RoboDK station: ME5286_Lab4_Serdoncillo_JustineJohnv1.rdk

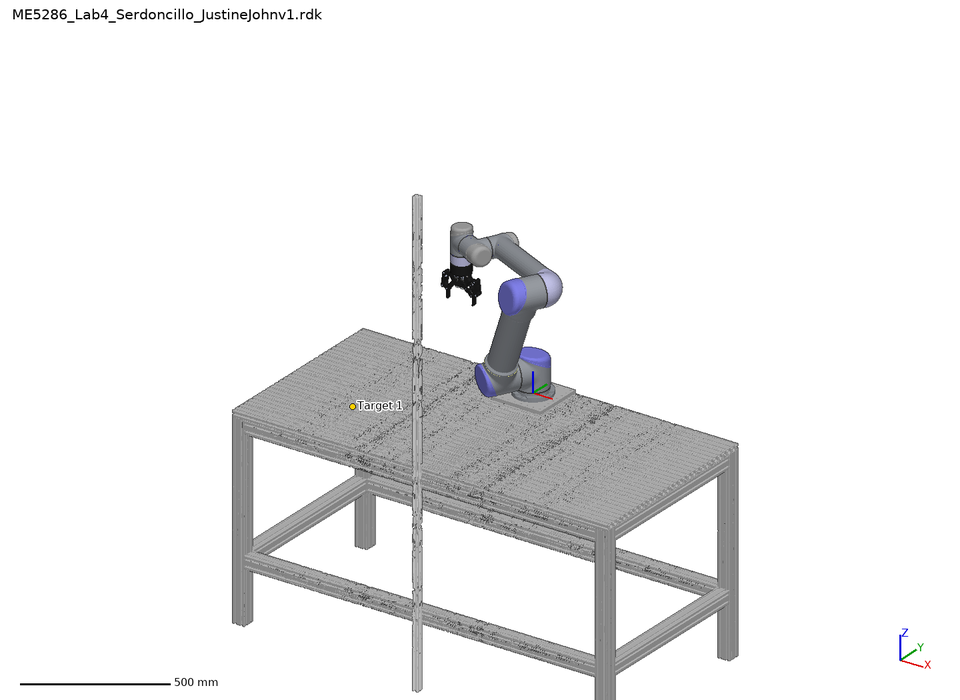
[picture v0: the station drawn from its stored meshes, robots at their saved joint values, targets as dots, program paths as lines]
Station ME5286_Lab4_Serdoncillo_JustineJohnv1 (saved by RoboDK 5.5.3). Poses are relative to the parent item; angles as X-Y-Z fixed-axis rotations.
  - frame UR5 Base at (0, 0, 0) mm
    - robot UR5: 6 axes, payload 5 kg, reach 850 mm, repeatability 0.1 mm, weight 18.4 kg
        modified DH rows (alpha deg, a mm, theta deg, d mm): 0, 0, 0, 89.2; 90, 0, 180, 0; 0, 425, 0, 0; 0, 392.43, 0, 109; -90, 0, 0, 93.65; 90, 0, 180, 82
        joint limits [-360, -360, -360, -360, -360, -360] to [360, 360, 360, 360, 360, 360]; home [0, -90, 90, 0, 90, 0]; saved at [-27.14, -115.32, 117.34, -92.04, -89.49, -26.91]
      - tool Gripper RobotiQ 85 Opened, TCP at (0, 0, 149.6) mm, size 147.4 x 146.8 x 75 mm
    - target Target 1 (Cartesian target) at (-388.22, -492.26, 39) mm, rotated rx 177.02 ry -0.73 rz 86.38 deg; joints [41.133, -63.138, 92.728, -116.961, -88.419, 44.733] of UR5
    - target Target 2 (Cartesian target) at (-388.22, -492.26, 39) mm, rotated rx -50 ry 58 rz -176 deg; joints [-116.508, -127.571, 233.195, -85.641, -85.367, -117.262] of UR5
  - object table_base_setup at (0, 0, 0) mm, rotated rx 0 ry 0 rz -90 deg, size 1524 x 762 x 800.1 mm, geometry from table_base_setup.STEP
  - object 6ft_beam_table at (0, -675, 1000) mm, size 25.4 x 25.4 x 1828.8 mm, geometry from 6ft_beam_table.IGS
  - Python program ME5286_Lab4_Task_Serdoncillo_JustineJohnv3 (listed below)

--- Python program ME5286_Lab4_Task_Serdoncillo_JustineJohnv3 ---
# This macro shows an example of running a program on the robot using the Python API (online programming)
# More information about the RoboDK API appears here:
# https://robodk.com/doc/en/RoboDK-API.html
import sys
sys.path.append("C:\RoboDK\Python")
#############################################################
from robolink import *    # API to communicate with RoboDK
from robodk import *      # robodk robotics toolbox
RDK = Robolink()
robot = RDK.ItemUserPick('Select a robot', ITEM_TYPE_ROBOT)
if not robot.Valid():
    raise Exception('No robot selected or available')
RUN_ON_ROBOT = False
if RDK.RunMode() != RUNMODE_SIMULATE:
    RUN_ON_ROBOT = False
if RUN_ON_ROBOT:
    # Connect to the robot using default IP
    success = robot.Connect() # Try to connect once
    status, status_msg = robot.ConnectedState()
    if status != ROBOTCOM_READY:
        # Stop if the connection did not succeed
        print(status_msg)
        raise Exception("Failed to connect: " + status_msg)
    # This will set to run the API programs on the robot and the simulator (online programming)
    RDK.setRunMode(RUNMODE_RUN_ROBOT)
joints_ref = robot.Joints()
target_ref = robot.Pose()
pos_ref = target_ref.Pos()
robot.setPoseFrame(robot.PoseFrame())
robot.setPoseTool(robot.PoseTool())
###################################################################
## JJ Code down below
import numpy as np
###################################################################
linspeed = [250]
linaccel = [200]
joispeed = [15]
joiaccel = [60]
robot.setSpeed(50) # Set linear speed in mm/s
robot.setAcceleration(100) # Set acceleration in mm/s
robot.setSpeedJoints(15) # Set joint speed in deg/s
robot.setAccelerationJoints(60) # Set joint accel in deg/s^2
robot.setZoneData(2) # Set blending radius in mm
##################################################################
gripper_force = [127,127,127,127]
gripper_speed = [ 50, 50, 50, 50]
pos = np.array([ [0, 0, 0, 0] , [0, 9, 6, 3] ]) * 25.4
##################################################################
# input values here
tray_og =  [-389.00 ,-494.00] # origin of the tray in x,y,z
chuck_og = [-322.00 ,  40.00] # origin of the chuck in x,y,z
#-388.22 ,-492.26
#-322.39 ,  39.89: old chuck_og and not centered
#-320.37 ,  39.9
#deg = [130,122,4] # ideal orientation
#deg = [-180,0,4] # from Lab 3 but hitting other components
#deg = [-176.79,-1.10,-89.55]
deg = [-180,0,-90]
tray_z  = np.array([39,50,43,38]) + 33 # Lab 3 has z=70 but these measurements s
chuck_z = np.array([140,185,225,227]) + 40 # 2 and 3 not sure

twist = [False,True,False,True]
#twist = [False, False, False, False]
#twist_num = [10,7]
twist_num = [6,3]
twist_torque = [3,2]
#############################################
theta_1 = 0
theta_2 = np.pi
cB = np.cos(theta_1)
sB = np.sin(theta_1)
cC = np.cos(theta_2)
sC = np.sin(theta_2)
TB = tray_og.copy()
TC = chuck_og.copy()
RTAB = np.array([[cB,-sB,TB[0]],[sB,cB,TB[1]],[0,0,1]])
RTAC = np.array([[cC,-sC,TC[0]],[sC,cC,TC[1]],[0,0,1]])

tray   = np.zeros((4,6))
chuck  = np.zeros((4,6))
tray[:,3] = deg[0]
tray[:,4] = deg[1]
tray[:,5] = deg[2]
chuck[:,0] = TC[0]
chuck[:,1] = TC[1]
chuck[:,3] = deg[0]
chuck[:,4] = deg[1]
chuck[:,5] = deg[2]
for j in range(4):
  P1B = np.array([[pos[0,j]],[pos[1,j]],[1]])
  P1A = RTAB @ P1B
  tray[j,0] = P1A[0]
  tray[j,1] = P1A[1]
  tray[j,2] = tray_z[j]
  chuck[j,2] = chuck_z[j]
tray_up = tray.copy()
tray_up[:,2] += 30
chuck_up = chuck.copy()
chuck_up[:,2] += 110

#twist_before = np.zeros((2,6))
'''
twist_before[0] = chuck[1]
twist_before[1] = chuck[3]
twist_after = twist_before.copy()
twist_after[:,5] = 90
'''
twist_before = [-27.14,-115.32,117.34,-92.04,-89.49,-206.91]
#twist_before[0] = [-27.14,-115.32,117.34,-92.04,-89.49,-206.91]
twist_after = twist_before.copy()
twist_after[5] += 180

twist_count = 0

###################################################################
''' Do manual stuff rn '''
home = [0, -90, 0, -90, 0, 0]
robot.MoveJ(home)
safe = [35.30,-90.35,87.92,-90.26,-90.32,-43.42]
robot.MoveJ(safe)

robot.RunCodeCustom('unclamp()',INSTRUCTION_INSERT_CODE)
#robot.RunCodeCustom('clamp()',INSTRUCTION_INSERT_CODE)
#range(4)

for i in np.arange(0,2):
    robot.RunCodeCustom('rq_set_force(%i)' %gripper_force[i], INSTRUCTION_CALL_PROGRAM)
    robot.RunCodeCustom('rq_set_speed(%i)' %gripper_speed[i], INSTRUCTION_CALL_PROGRAM)
    robot.MoveL(xyzrpw_2_pose(tray[i]))
    robot.RunCodeCustom('rq_close_and_wait()',INSTRUCTION_CALL_PROGRAM)
    robot.MoveL(xyzrpw_2_pose(tray_up[i]))
    robot.MoveL(xyzrpw_2_pose(chuck_up[i]))
    robot.MoveL(xyzrpw_2_pose(chuck[i]))
    #robot.RunCodeCustom('sleep(10)',INSTRUCTION_CALL_PROGRAM)
    if i != 3:
        robot.RunCodeCustom('rq_open_and_wait()',INSTRUCTION_CALL_PROGRAM)
    if twist[i] == True:
        for tnum in range(twist_num[twist_count]):
            robot.MoveJ(twist_before)
            #robot.MoveJ(xyzrpw_2_pose(twist_before[twist_count]))
            robot.RunCodeCustom('rq_close_and_wait()',INSTRUCTION_CALL_PROGRAM)
            robot.MoveJ(twist_after)
            #robot.MoveJ(xyzrpw_2_pose(twist_after[twist_count]))
            robot.RunCodeCustom('rq_open_and_wait()',INSTRUCTION_CALL_PROGRAM)
        robot.RunCodeCustom('tighten_torque(%i,0,1.57,2,2,1,100,100,50)' %twist_torque[twist_count],INSTRUCTION_INSERT_CODE)
        twist_count += 1
    if i == 0:
        robot.RunCodeCustom('clamp()',INSTRUCTION_INSERT_CODE)
    elif i == 3:
        robot.RunCodeCustom('unclamp()',INSTRUCTION_INSERT_CODE)
    robot.MoveL(xyzrpw_2_pose(chuck[i]))
    robot.MoveL(xyzrpw_2_pose(chuck_up[i]))
    #robot.RunCodeCustom('sleep(10)',INSTRUCTION_CALL_PROGRAM)

#robot.MoveJ(safe)
#robot.MoveJ(home)
